PROGRAM MAIN
VAR
END_VAR

SolenoidPairA();

fb_4PortViciValve_01(iAdress:=1);

(* Following execution of all the programs, set the first pass false *)
g_xFirstPass := FALSE;

END_PROGRAM

(* stored: Version 1.1.0.1, ProductVersion 3.1.4022.18
   POU MAIN: Id {92caf389-36e1-4cad-84b9-376141bd147e}, SpecialFunc None *)
